// TIA Portal V17 export
// export: Created 2023-12-05T13:40:22.2677941Z, ExportSetting WithDefaults, DisplayName Totally Integrated Automation Portal, DisplayVersion V17, DisplayName TIA Portal Openness, DisplayVersion V17, DisplayName TIA Portal Version Control Interface, DisplayVersion V17, DisplayName SINAMICS Startdrive Advanced, DisplayVersion V17, DisplayName SINAMICS Startdrive G130, G150, S120, S150, SINAMICS MV, S210, DisplayVersion V17, DisplayName SINAMICS Startdrive G110M, G120, G120C, G120D, G120P, G115D, DisplayVersion V17, DisplayName STEP 7 Professional, DisplayVersion V17, DisplayName STEP 7 Safety, DisplayVersion V17, DisplayName WinCC Professional, DisplayVersion V17
FUNCTION "FC515 Movement from SB for IC" : Void   // FC515, LAD
{ S7_Optimized_Access := 'TRUE' }
VERSION : 0.1
// LM Created 2023_06_28
// Intervention request check for SB movement
// stored: AutoNumber false, IsIECCheckEnabled false, SetENOAutomatically false, UDAEnableTagReadback false
   VAR_INPUT
      "at WP" : Bool;   // Working Position Sensor
      "at PP" : Bool;   // Parking Position Sensor
      "to WP/PP manu" : "cylinder";   // Working/Parking Position in Manual
      GCYLSensorTime : Time;
   END_VAR
   VAR_IN_OUT
      GeneralStruct : "MoveAlarmGeneral";
      SingleStruct : "MoveAlarmSingle";
   END_VAR
BEGIN

REGION Network 2: Movement to working in manual mode
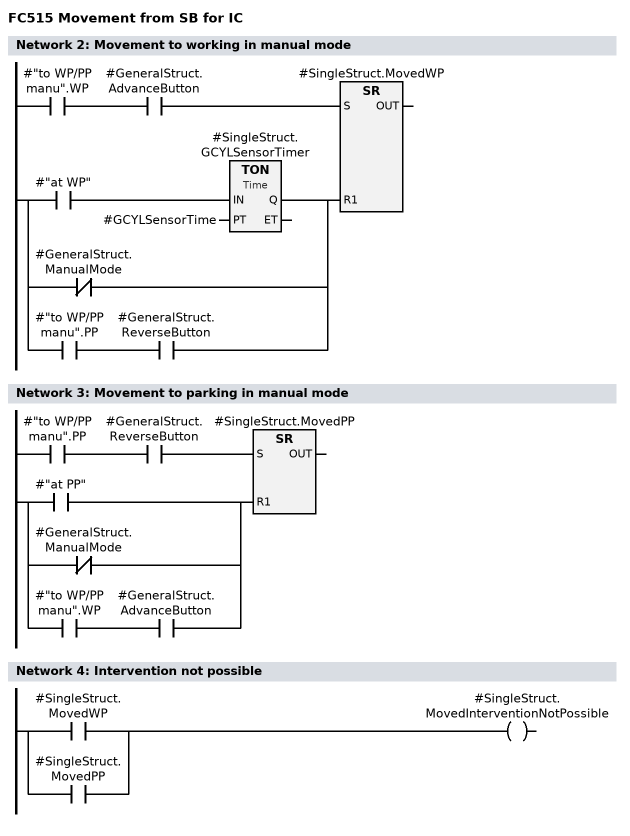
   RUNG wire#powerrail
      Contact( #"to WP/PP manu".WP )
      Contact( #GeneralStruct.AdvanceButton )
      S_SR(operand := #SingleStruct.MovedWP, r1 := wire#w1)
   END_RUNG
   RUNG wire#powerrail
      Contact( #"at WP" )
      { S7_Templates := "time_type := Time" } #SingleStruct.GCYLSensorTimer.TON(pt := #GCYLSensorTime, et =>)
   END_RUNG wire#w1
   RUNG wire#powerrail
      I_Contact( #GeneralStruct.ManualMode )
   END_RUNG wire#w1
   RUNG wire#powerrail
      Contact( #"to WP/PP manu".PP )
      Contact( #GeneralStruct.ReverseButton )
   END_RUNG wire#w1
   // the same network as SCL:
   #SingleStruct.GCYLSensorTimer.TON(IN := #"at WP", PT := #GCYLSensorTime);
   IF #"to WP/PP manu".WP AND #GeneralStruct.AdvanceButton THEN
       #SingleStruct.MovedWP := TRUE;   // SR flip-flop
   END_IF;
   IF #SingleStruct.GCYLSensorTimer.Q OR NOT #GeneralStruct.ManualMode OR (#"to WP/PP manu".PP AND #GeneralStruct.ReverseButton) THEN
       #SingleStruct.MovedWP := FALSE;
   END_IF;
END_REGION

REGION Network 3: Movement to parking in manual mode
   RUNG wire#powerrail
      Contact( #"to WP/PP manu".PP )
      Contact( #GeneralStruct.ReverseButton )
      S_SR(operand := #SingleStruct.MovedPP, r1 := wire#w1)
   END_RUNG
   RUNG wire#powerrail
      Contact( #"at PP" )
   END_RUNG wire#w1
   RUNG wire#powerrail
      I_Contact( #GeneralStruct.ManualMode )
   END_RUNG wire#w1
   RUNG wire#powerrail
      Contact( #"to WP/PP manu".WP )
      Contact( #GeneralStruct.AdvanceButton )
   END_RUNG wire#w1
   // the same network as SCL:
   IF #"to WP/PP manu".PP AND #GeneralStruct.ReverseButton THEN
       #SingleStruct.MovedPP := TRUE;   // SR flip-flop
   END_IF;
   IF #"at PP" OR NOT #GeneralStruct.ManualMode OR (#"to WP/PP manu".WP AND #GeneralStruct.AdvanceButton) THEN
       #SingleStruct.MovedPP := FALSE;
   END_IF;
END_REGION

REGION Network 4: Intervention not possible
   RUNG wire#powerrail
      Contact( #SingleStruct.MovedWP )
      wire#w1
      Coil( #SingleStruct.MovedInterventionNotPossible )
   END_RUNG
   RUNG wire#powerrail
      Contact( #SingleStruct.MovedPP )
   END_RUNG wire#w1
   // the same network as SCL:
   #SingleStruct.MovedInterventionNotPossible := #SingleStruct.MovedWP OR #SingleStruct.MovedPP;
END_REGION
END_FUNCTION
